// TIA Portal V18 export
FUNCTION_BLOCK "SR_CLK"   // FB9, FBD
{ S7_Optimized_Access := 'TRUE' }
VERSION : 0.1
// stored: AutoNumber true, IsIECCheckEnabled false, IsRetainMemResEnabled false, MemoryReserve 100, SetENOAutomatically false, UDAEnableTagReadback false
   VAR_INPUT
      CLK : Bool;
   END_VAR
   VAR_IN_OUT
      Q : Bool;
   END_VAR
   VAR
      mem_R : Bool;
      mem_S : Bool;
   END_VAR
   VAR_TEMP   // added for the SCL form of the ladder/FBD networks
      _w1 : Bool;
      _w2 : Bool;
   END_VAR
BEGIN

REGION Network 1
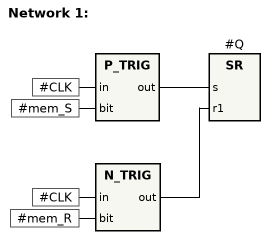
   #_w1 := #CLK AND NOT #mem_S;   // rising edge
   #mem_S := #CLK;
   #_w2 := NOT #CLK AND #mem_R;   // falling edge
   #mem_R := #CLK;
   IF #_w1 THEN
       #Q := TRUE;   // SR flip-flop
   END_IF;
   IF #_w2 THEN #Q := FALSE; END_IF;
END_REGION
END_FUNCTION_BLOCK
